Staubli VAL3: loadEditTraj.pgx

program loadEditTraj(string x_sName)
  local num i
  local num l_nIndex
  local string l_sPath
begin
end
